TEXTLIST TL_MessageList
  7 = 'eCONVEYOR_1_AT_TRANSFER_POINT'
  8 = 'eCONVEYOR_1_RESUMING_OPERATION'
  9 = 'eCONVEYOR_2_AT_TRANSFER_POINT'
  10 = 'eCONVEYOR_2_RESUMING_OPERATION'
  11 = 'eCONVEYOR_3_AT_TRANSFER_POINT'
  12 = 'eCONVEYOR_3_RESUMING_OPERATION'
  13 = 'eCONVEYOR_4_AT_TRANSFER_POINT'
  14 = 'eCONVEYOR_4_RESUMING_OPERATION'
  15 = ''
  16 = ''
  17 = ''
   = ''
END_TEXTLIST

(* stored: Version 1.1.0.1, ProductVersion 3.1.4022.16
   TextList TL_MessageList: Id {7125f7e7-b921-4f85-866b-48be0acb9ad8} *)
